FUNCTION ATT_TO_IO : ST_PMPS_Attenuator_IO
VAR_INPUT
    Att : ST_PMPS_Attenuator;
END_VAR
VAR
END_VAR

ATT_TO_IO.nAtt := Att.nAtt;
ATT_TO_IO.xAttOK := Att.xAttOK;

END_FUNCTION

(* stored: Version 1.1.0.1, ProductVersion 3.1.4022.18
   POU ATT_TO_IO: Id {18b528b7-b147-4652-8142-65b2d820ca1f}, SpecialFunc None *)
